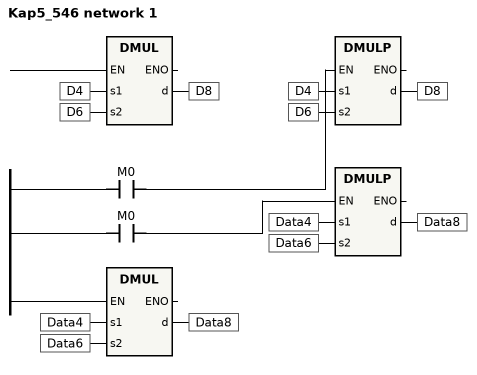
(* [picture p48: structured ladder/FBD of Kap5_546, networks 1 to 1] *)
(* network 1 *)
DMUL(TRUE, D4, D6, D8);
DMUL(TRUE, Data4, Data6, Data8);
DMULP(M0, D4, D6, D8);
DMULP(M0, Data4, Data6, Data8);
END_PROGRAM

PROGRAM Kap5_547
VAR
  Data1 : INT;
  Data2 : INT;
  Data3 : ARRAY [0..1] OF INT;
END_VAR
(* structured ladder/FBD written out as ST: instructions are called as NAME(EN, inputs, outputs); _pN, _eN, _tN stand for wires *)
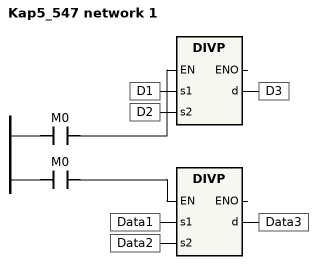
(* network 1 *)
DIVP(M0, D1, D2, D3);
DIVP(M0, Data1, Data2, Data3);
END_PROGRAM

PROGRAM Kap5_548
VAR
  Data4 : DINT;
  Data6 : DINT;
  Data8 : ARRAY [0..1] OF DINT;
END_VAR
(* structured ladder/FBD written out as ST: instructions are called as NAME(EN, inputs, outputs); _pN, _eN, _tN stand for wires *)
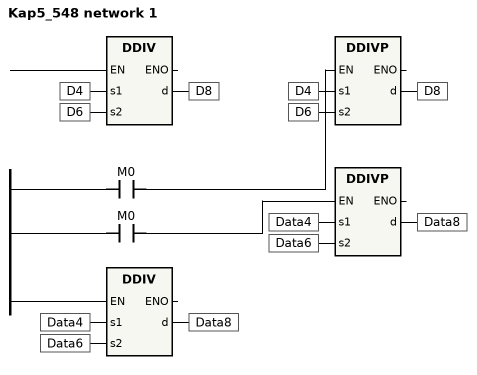
(* network 1 *)
DDIV(TRUE, D4, D6, D8);
DDIV(TRUE, Data4, Data6, Data8);
DDIVP(M0, D4, D6, D8);
DDIVP(M0, Data4, Data6, Data8);
END_PROGRAM

PROGRAM Kap5_549
(* structured ladder/FBD written out as ST: instructions are called as NAME(EN, inputs, outputs); _pN, _eN, _tN stand for wires *)
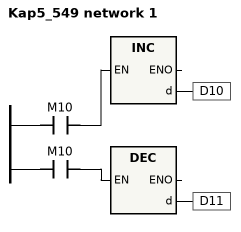
(* network 1 *)
INC(M10, D10);
DEC(M10, D11);
END_PROGRAM

PROGRAM Kap5_5410
(* structured ladder/FBD written out as ST: instructions are called as NAME(EN, inputs, outputs); _pN, _eN, _tN stand for wires *)
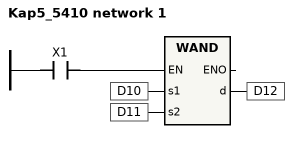
(* network 1 *)
WAND(X1, D10, D11, D12);
END_PROGRAM

PROGRAM Kap5_5411
(* structured ladder/FBD written out as ST: instructions are called as NAME(EN, inputs, outputs); _pN, _eN, _tN stand for wires *)
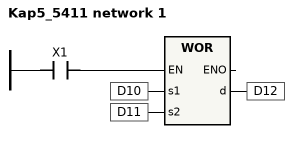
(* network 1 *)
WOR(X1, D10, D11, D12);
END_PROGRAM

PROGRAM Kap5_5412
(* structured ladder/FBD written out as ST: instructions are called as NAME(EN, inputs, outputs); _pN, _eN, _tN stand for wires *)
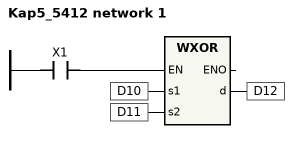
(* network 1 *)
WXOR(X1, D10, D11, D12);
END_PROGRAM

PROGRAM Kap5_5415
VAR
  Sammenlign_D0_100 : ARRAY [0..2] OF BOOL;
END_VAR
(* structured ladder/FBD written out as ST: instructions are called as NAME(EN, inputs, outputs); _pN, _eN, _tN stand for wires *)
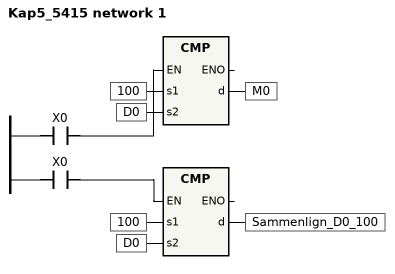
(* network 1 *)
CMP(X0, 100, D0, M0);
CMP(X0, 100, D0, Sammenlign_D0_100);
END_PROGRAM

PROGRAM Kap5_5416
VAR
  Sammenlign_D1_100_120 : ARRAY [0..2] OF BOOL;
END_VAR
(* structured ladder/FBD written out as ST: instructions are called as NAME(EN, inputs, outputs); _pN, _eN, _tN stand for wires *)
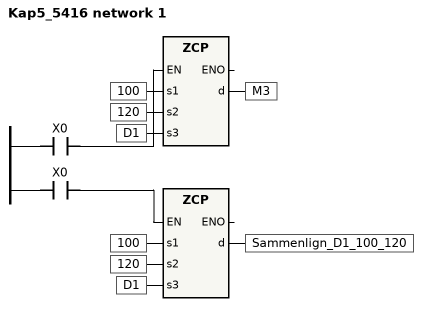
(* network 1 *)
ZCP(X0, 100, 120, D1, M3);
ZCP(X0, 100, 120, D1, Sammenlign_D1_100_120);
END_PROGRAM

PROGRAM Kap5_5417
(* structured ladder/FBD written out as ST: instructions are called as NAME(EN, inputs, outputs); _pN, _eN, _tN stand for wires *)
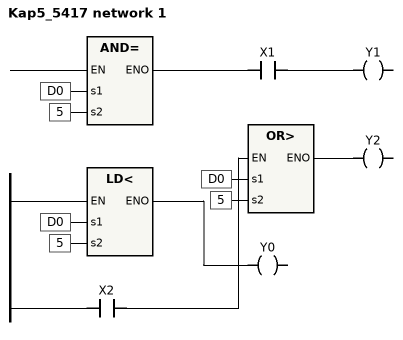
(* network 1 *)
_e1 := LD<(TRUE, D0, 5);
Y0 := _e1;
_e2 := AND=(TRUE, D0, 5);
Y1 := _e2 AND X1;
_e3 := OR>(X2, D0, 5);
Y2 := _e3;
END_PROGRAM

PROGRAM Kap5_5418
(* structured ladder/FBD written out as ST: instructions are called as NAME(EN, inputs, outputs); _pN, _eN, _tN stand for wires *)
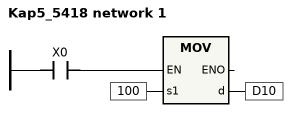
(* network 1 *)
MOV(X0, 100, D10);
END_PROGRAM

PROGRAM Kap5_5419
(* structured ladder/FBD written out as ST: instructions are called as NAME(EN, inputs, outputs); _pN, _eN, _tN stand for wires *)
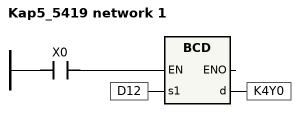
(* network 1 *)
BCD(X0, D12, K4Y0);
END_PROGRAM

PROGRAM Kap5_5420
(* structured ladder/FBD written out as ST: instructions are called as NAME(EN, inputs, outputs); _pN, _eN, _tN stand for wires *)
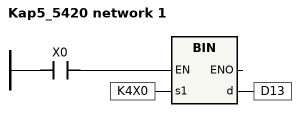
(* network 1 *)
BIN(X0, K4X0, D13);
END_PROGRAM

PROGRAM Kap5_5423
(* structured ladder/FBD written out as ST: instructions are called as NAME(EN, inputs, outputs); _pN, _eN, _tN stand for wires *)
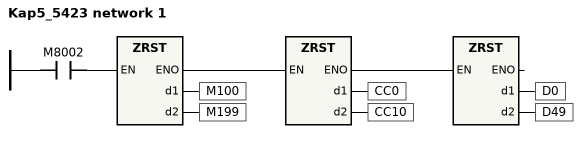
(* network 1 *)
_e1 := ZRST(M8002, M100, M199);
_e2 := ZRST(_e1, CC0, CC10);
ZRST(_e2, D0, D49);
END_PROGRAM

PROGRAM Kap5_5425
(* structured ladder/FBD written out as ST: instructions are called as NAME(EN, inputs, outputs); _pN, _eN, _tN stand for wires *)
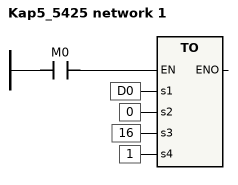
(* network 1 *)
TO(M0, D0, 0, 16, 1);
END_PROGRAM

PROGRAM Kap5_5426
(* structured ladder/FBD written out as ST: instructions are called as NAME(EN, inputs, outputs); _pN, _eN, _tN stand for wires *)
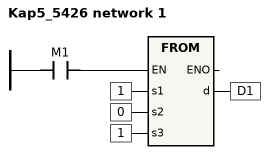
(* network 1 *)
FROM(M1, 1, 0, 1, D1);
END_PROGRAM

PROGRAM Kap5_5429_5430
VAR
  Var1 : INT;
  Var2 : INT;
  Var3 : DINT;
  Var4 : DINT;
  Var5 : DINT;
  Var6 : DINT;
  Var7 : REAL;
  Var8 : REAL;
  Var9 : REAL;
  Var10 : REAL;
  Var11 : REAL;
  Var12 : REAL;
  Var13 : REAL;
  Var14 : REAL;
  Ut1 : INT;
  Ut2 : DINT;
  Ut3 : DINT;
  Ut4 : REAL;
  Ut5 : REAL;
  Ut6 : REAL;
  Ut7 : REAL;
END_VAR
(* structured ladder/FBD written out as ST: instructions are called as NAME(EN, inputs, outputs); _pN, _eN, _tN stand for wires *)
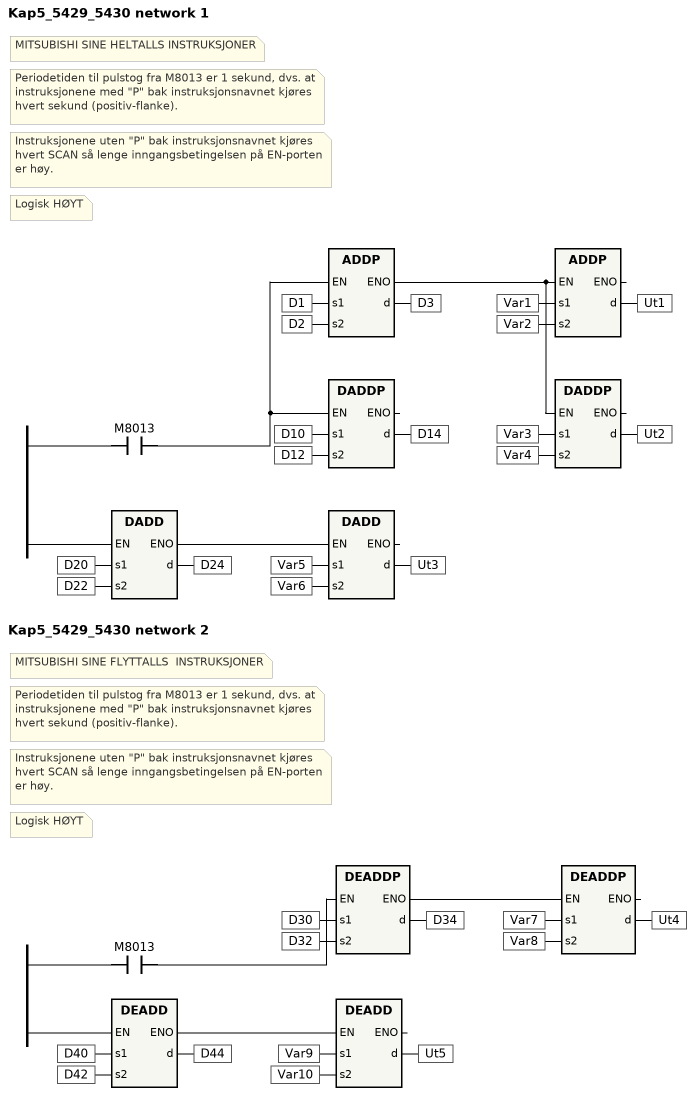
(* network 1 *)
(* MITSUBISHI SINE HELTALLS INSTRUKSJONER *)
(* Periodetiden til pulstog fra M8013 er 1 sekund, dvs. at instruksjonene med "P" bak instruksjonsnavnet kjøres hvert sekund (positiv-flanke). *)
(* Instruksjonene uten "P" bak instruksjonsnavnet kjøres hvert SCAN så lenge inngangsbetingelsen på EN-porten er høy. *)
(* Logisk HØYT *)
_e1 := ADDP(M8013, D1, D2, D3);
ADDP(_e1, Var1, Var2, Ut1);
DADDP(M8013, D10, D12, D14);
DADDP(_e1, Var3, Var4, Ut2);
_e2 := DADD(TRUE, D20, D22, D24);
DADD(_e2, Var5, Var6, Ut3);
(* network 2 *)
(* MITSUBISHI SINE FLYTTALLS  INSTRUKSJONER *)
(* Periodetiden til pulstog fra M8013 er 1 sekund, dvs. at instruksjonene med "P" bak instruksjonsnavnet kjøres hvert sekund (positiv-flanke). *)
(* Instruksjonene uten "P" bak instruksjonsnavnet kjøres hvert SCAN så lenge inngangsbetingelsen på EN-porten er høy. *)
(* Logisk HØYT *)
_e1 := DEADDP(M8013, D30, D32, D34);
DEADDP(_e1, Var7, Var8, Ut4);
_e2 := DEADD(TRUE, D40, D42, D44);
DEADD(_e2, Var9, Var10, Ut5);
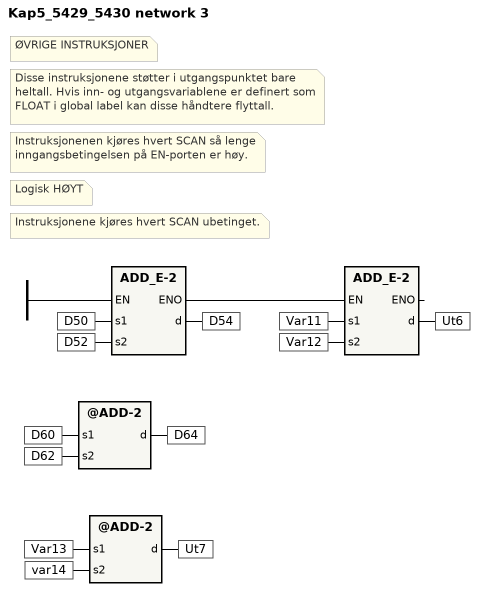
(* network 3 *)
(* ØVRIGE INSTRUKSJONER *)
(* Disse instruksjonene støtter i utgangspunktet bare heltall. Hvis inn- og utgangsvariablene er definert som FLOAT i global label kan disse håndtere flyttall. *)
(* Instruksjonenen kjøres hvert SCAN så lenge inngangsbetingelsen på EN-porten er høy. *)
(* Logisk HØYT *)
(* Instruksjonene kjøres hvert SCAN ubetinget. *)
_e1 := ADD_E(TRUE, D50, D52, D54);
ADD_E(_e1, Var11, Var12, Ut6);
D64 := @ADD-2(D60, D62);
Ut7 := @ADD-2(Var13, var14);
END_PROGRAM

PROGRAM Kap3_327
(* structured ladder/FBD written out as ST: instructions are called as NAME(EN, inputs, outputs); _pN, _eN, _tN stand for wires *)
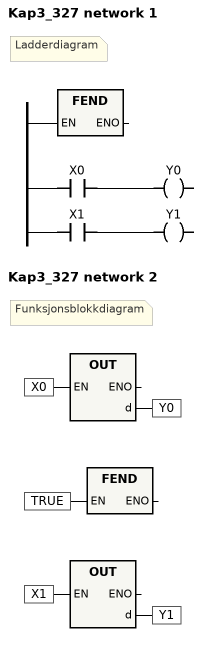
(* network 1 *)
(* Ladderdiagram *)
Y0 := X0;
FEND(TRUE);
Y1 := X1;
(* network 2 *)
(* Funksjonsblokkdiagram *)
OUT(X0, Y0);
FEND(TRUE);
OUT(X1, Y1);
END_PROGRAM

PROGRAM Kap4_423
(* structured ladder/FBD written out as ST: instructions are called as NAME(EN, inputs, outputs); _pN, _eN, _tN stand for wires *)
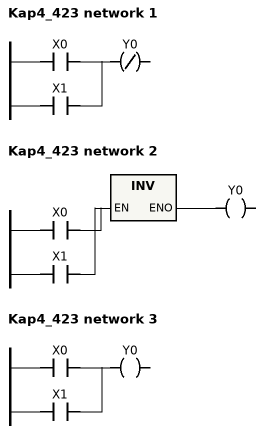
(* network 1 *)
Y0 := NOT (X0 OR X1);
(* network 2 *)
_e1 := INV(X0 OR X1);
Y0 := _e1;
(* network 3 *)
Y0 := X0 OR X1;
END_PROGRAM

PROGRAM Kap4_484
VAR
  Start : BOOL;
  Stopp : BOOL;
  Startflagg : BOOL;
  Alarm : BOOL;
  Kvittering : BOOL;
  KvittertAlarm : BOOL;
  Motorvern : BOOL;
  Feil : BOOL;
  Motor : BOOL;
  AlarmLampe : BOOL;
END_VAR
(* structured ladder/FBD written out as ST: instructions are called as NAME(EN, inputs, outputs); _pN, _eN, _tN stand for wires *)
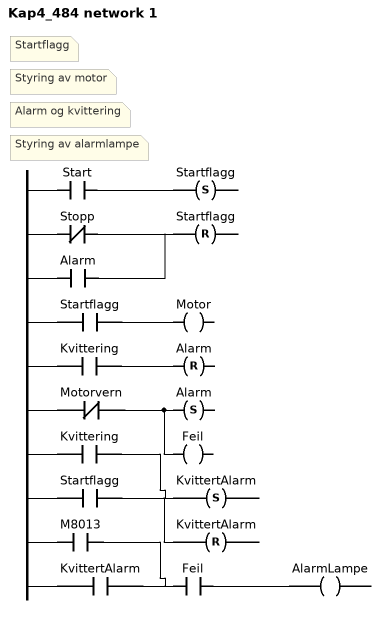
(* network 1 *)
(* Startflagg *)
(* Styring av motor *)
(* Alarm og kvittering *)
(* Styring av alarmlampe *)
SET(Start, Startflagg);
RST((NOT Stopp) OR Alarm, Startflagg);
Motor := Startflagg;
RST(Kvittering, Alarm);
_p1 := NOT Motorvern;
SET(_p1, Alarm);
Feil := _p1;
SET(Kvittering, KvittertAlarm);
RST(Startflagg, KvittertAlarm);
AlarmLampe := (M8013 OR KvittertAlarm) AND Feil;
END_PROGRAM

PROGRAM Kap5_5428
VAR
  PV : WORD;
  CV : WORD;
END_VAR
(* structured ladder/FBD written out as ST: instructions are called as NAME(EN, inputs, outputs); _pN, _eN, _tN stand for wires *)
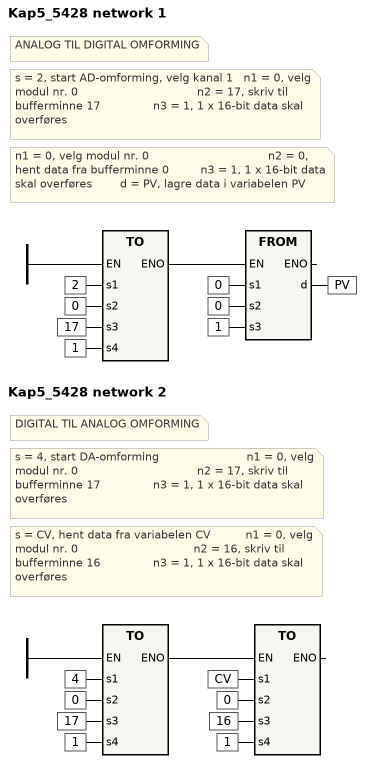
(* network 1 *)
(* ANALOG TIL DIGITAL OMFORMING *)
(* s = 2, start AD-omforming, velg kanal 1   n1 = 0, velg modul nr. 0                                  n2 = 17, skriv til bufferminne 17               n3 = 1, 1 x 16-bit data skal overføres *)
(* n1 = 0, velg modul nr. 0                                  n2 = 0, hent data fra bufferminne 0         n3 = 1, 1 x 16-bit data skal overføres        d = PV, lagre data i variabelen PV *)
_e1 := TO(TRUE, 2, 0, 17, 1);
FROM(_e1, 0, 0, 1, PV);
(* network 2 *)
(* DIGITAL TIL ANALOG OMFORMING *)
(* s = 4, start DA-omforming                         n1 = 0, velg modul nr. 0                                  n2 = 17, skriv til bufferminne 17               n3 = 1, 1 x 16-bit data skal overføres *)
(* s = CV, hent data fra variabelen CV          n1 = 0, velg modul nr. 0                                 n2 = 16, skriv til bufferminne 16               n3 = 1, 1 x 16-bit data skal overføres *)
_e1 := TO(TRUE, 4, 0, 17, 1);
TO(_e1, CV, 0, 16, 1);
END_PROGRAM

PROGRAM Kap3_334
(* structured ladder/FBD written out as ST: instructions are called as NAME(EN, inputs, outputs); _pN, _eN, _tN stand for wires *)
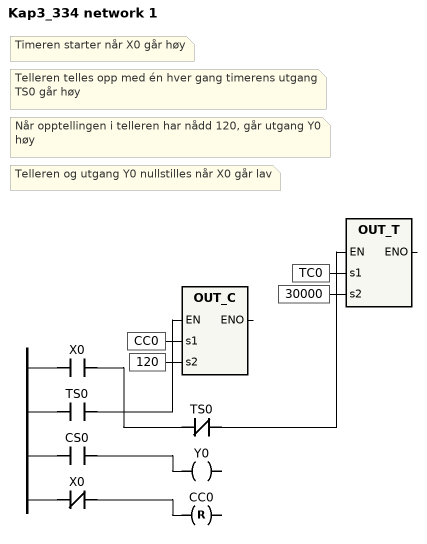
(* network 1 *)
(* Timeren starter når X0 går høy *)
(* Telleren telles opp med én hver gang timerens utgang TS0 går høy *)
(* Når opptellingen i telleren har nådd 120, går utgang Y0 høy *)
(* Telleren og utgang Y0 nullstilles når X0 går lav *)
OUT_T(X0 AND NOT TS0, TC0, 30000);
OUT_C(TS0, CC0, 120);
Y0 := CS0;
RST(NOT X0, CC0);
END_PROGRAM
